FUNCTION_BLOCK SSC_TransferWorkpieceTo_RampEnd EXTENDS SSC_MoveWorkpiece_Base
VAR_INPUT
END_VAR
VAR_OUTPUT
END_VAR
VAR
	// (EProcessVariables.PicAlpha_AtPos3 = TRUE) AND ((EProcessVariables.PicAlpha_HoldingWorkpiece = FALSE) AND (EProcessVariables.PicAlpha_CylinderExtended = FALSE))
	m_compExpr233: ComparisonExpression(EProcessVariables.PicAlpha_AtPos3, EComparisonType.equals, EDataType.binary, TRUE, 0, '', TRUE);
	m_compExpr235: ComparisonExpression(EProcessVariables.PicAlpha_HoldingWorkpiece, EComparisonType.equals, EDataType.binary, FALSE, 0, '', TRUE);
	m_compExpr237: ComparisonExpression(EProcessVariables.PicAlpha_CylinderExtended, EComparisonType.equals, EDataType.binary, FALSE, 0, '', TRUE);
	m_boolExpr238: BoolExpression(m_compExpr235, EBoolOperation.and_op, m_compExpr237);
	m_precondition: BoolExpression(m_compExpr233, EBoolOperation.and_op, m_boolExpr238);
	
	// TRUE
	m_postcondition: ValueExpression(EDataType.binary, TRUE, 0, '', TRUE);
	
	m_timer: TON;
	m_passby : BOOL;
END_VAR

SUPER^();

METHOD PROTECTED  AtTarget : BOOL
VAR_INPUT
END_VAR

IF m_ptrSSC^.WPAtRampEnd THEN
	m_passby := TRUE;
END_IF

IF m_passby THEN
	m_timer(IN := TRUE, PT := T#200MS);
	IF m_timer.Q THEN
		m_timer(IN := FALSE);
		m_passby := FALSE;
		AtTarget := TRUE;
	END_IF
END_IF
END_METHOD

METHOD FB_init : BOOL
VAR_INPUT
	bInitRetains : BOOL; // if TRUE, the retain variables are initialized (warm start / cold start)
	bInCopyCode : BOOL;  // if TRUE, the instance afterwards gets moved into the copy code (online change)
	
	i_ptrSSC: POINTER TO SmallSortingConveyor;
END_VAR
m_ptrSSC := i_ptrSSC;

m_id := EPrimitives.SSC_TransferWorkpieceTo_RampEnd;
m_timeout := T#200S;

Precondition := m_precondition;
Postcondition := m_postcondition;
END_METHOD

END_FUNCTION_BLOCK

(* stored: Version 1.1.0.1
   POU SSC_TransferWorkpieceTo_RampEnd: Id {25f88497-3c36-4144-842f-a645a1cb1aa8}, SpecialFunc None
   Method AtTarget: Id {8fe1faf6-e1a9-4e1c-a42f-071bec6c080d}
   Method FB_init: Id {33d68a85-5930-40b1-a6e2-864d50cacecf} *)
